(* PLC project Tc2_Utilities.FB_GetTimeZoneInformation Demo, tc3-libraries-kb TwinCAT 3.1 *)
(* stored: creationDateTime 2026-05-11T00:00:00, modificationDateTime 2026-05-11T00:00:00 *)

PROGRAM P_Demo_FB_GetTimeZoneInformation
  VAR
    fbFB_GetTimeZoneInformation : FB_GetTimeZoneInformation;  (* FB_GetTimeZoneInformation 实例 *)
    bRead : BOOL := FALSE;
    stTz : TIME_ZONE_INFORMATION;
    bDstNow : BOOL;
    bBusy_ : BOOL;
    bErrFlag : BOOL;
    nErrCode : UDINT;
  END_VAR

// =============================================================================
// 场景：读机器时区供 UTC 转换使用。
// 价值：标准 ADS 调用替代手工读注册表。
// 验证：改 bRead := TRUE，观察 stTz.Bias 与 Windows 控制面板时区一致；bDstNow 反映当前是否夏令时。
// 验证步骤：
//   1. 右键 PLC 项目 → Import PLCopenXML → 选本文件
//   2. 引用 Tc2_Utilities（References → Add library）
//   3. 编译 → 登录 → 运行；按上方『验证』行的指示在线写值观察
// =============================================================================

fbFB_GetTimeZoneInformation(
    sNetID := '', bExecute := bRead, tTimeout := DEFAULT_ADS_TIMEOUT,
    tzInfo => stTz, bDST => bDstNow,
    bBusy => bBusy_, bErr => bErrFlag, nErrId => nErrCode
);
END_PROGRAM
